FUNCTION Convert_SINT_TO_DINT : Hresult
VAR_INPUT
	in : SINT;
	out : REFERENCE TO DINT;
END_VAR
VAR
	converted : DINT;
END_VAR

converted := SINT_TO_DINT(in);

IF (DINT_TO_SINT(converted) <> in) THEN
	Convert_SINT_TO_DINT := INCOMPATIBLE;
	RETURN;
END_IF

out := converted;

END_FUNCTION

(* stored: Version 1.1.0.1, ProductVersion 3.1.4024.12
   POU Convert_SINT_TO_DINT: Id {f196a711-57b7-4de5-a39c-51c96ca5344b}, SpecialFunc None *)
